(*
Casts I_Arg as I_RealArg
*)
FUNCTION IArgToIRealtArg : Result
VAR_INPUT
	iArg		: I_Arg;
END_VAR
VAR_OUTPUT
	iVal		: I_RealArg;
END_VAR

IF __QUERYINTERFACE(iArg, iVal) THEN
	IArgToIRealtArg := Ok;
END_IF

END_FUNCTION

(* stored: Version 1.1.0.1
   POU IArgToIRealtArg: Id {6990d5d4-7f95-460d-b805-d7b0f1d0f775}, SpecialFunc None *)
